Omron CX-Programmer project NewProject (CX-Programmer 9.61)

# PLC Rubber_Sheet_thickness_control: CP1H XA

## Global symbols (name address type ; comment)
0.00 BOOL  ; Autostart
0.01 BOOL  ; Autostop
0.02 BOOL  ; Emergency
0.03 BOOL  ; Automode
0.04 BOOL  ; Emergency
0.10 BOOL  ; HMI1
0.11 BOOL  ; HMI2
0.12 BOOL  ; HMI3
0.13 BOOL  ; HMI4
100.00 BOOL  ; Auto_start_HMI
100.02 BOOL  ; PB_LAMP_GREEN
100.03 BOOL  ; PB_LAMP_RED
100.04 BOOL  ; Tipis_kiri
100.05 BOOL  ; Tebal_kiri
100.06 BOOL  ; Tipis _kanan
100.07 BOOL  ; Tebal_kanan
101.00 BOOL  ; TL_RED
101.01 BOOL  ; TL_YELLOW
101.02 BOOL  ; TL_GREEN
200 CHANNEL  ; Analog input 1
200.00 BOOL  ; Autostart_HMI
200.10 BOOL  ; EMO_AL
201 CHANNEL  ; Analog input 2
C0 CHANNEL  ; TIME
C0000 BOOL  ; COUNTER_1
D0 CHANNEL  ; SET_TIPIS_KIRI
D1 CHANNEL  ; SET_TEBAL_KIRI
D2 CHANNEL  ; SET_TIPIS_KANAN
D300 CHANNEL  ; SET_TEBAL_KANAN
D3010 CHANNEL  ; scalling 2
D310 CHANNEL  ; scalling 2
D400 CHANNEL  ; Output A
D410 CHANNEL  ; output B
D420 CHANNEL  ; output A
D5 CHANNEL  ; Scalled Ouput 0
H0.00 BOOL  ; TIPKIR
H0.01 BOOL  ; TEBKIR
H0.02 BOOL  ; TIPKAN
H0.03 BOOL  ; TEBKAN
H0.04 BOOL  ; TIPIS
H0.05 BOOL  ; TEBAL
H0.09 BOOL  ; TIPIS
H0.10 BOOL  ; TEBAL
H0.11 BOOL  ; HMI_Left thin adjust (button)
H0.12 BOOL  ; HMI_Left thick adjust (button)
H0.13 BOOL  ; HMI_Right thin adjust (button)
H0.14 BOOL  ; HMI_Right thick adjust (button)
H0.15 BOOL  ; reset timer
H100.00 BOOL  ; HOLD_Auto Start
H100.15 BOOL  ; reset timer
H200.01 BOOL  ; EMO_AL
H200.02 BOOL  ; TIPIS
H200.03 BOOL  ; TEBAL
T0000 BOOL  ; TIPKIR
T0001 BOOL  ; TEBKIR
T0002 BOOL  ; TIPKAN
T0003 BOOL  ; TEBKAN
T0004 BOOL  ; TIPIS
T0005 BOOL  ; TEBAL
T0006 BOOL  ; T_LIMIT
T0007 BOOL  ; T_LIMIT
T0008 BOOL  ; T_LIMIT
T0009 BOOL  ; T_LIMIT
T0010 BOOL  ; T_LIMIT
T0011 BOOL  ; T_LIMIT
W0 CHANNEL  ; TIPKIR
W1 CHANNEL  ; TEBKIR
W2 CHANNEL  ; TIPKAN
W3 CHANNEL  ; TEBKAN
W4 CHANNEL  ; TIPIS
W5 CHANNEL  ; TEBAL
W6 CHANNEL  ; TIME

## Program NewProgram1 (cyclic task 0)
Local symbols
TEBAL BOOL

### Section MAIN
; READ SENSOR

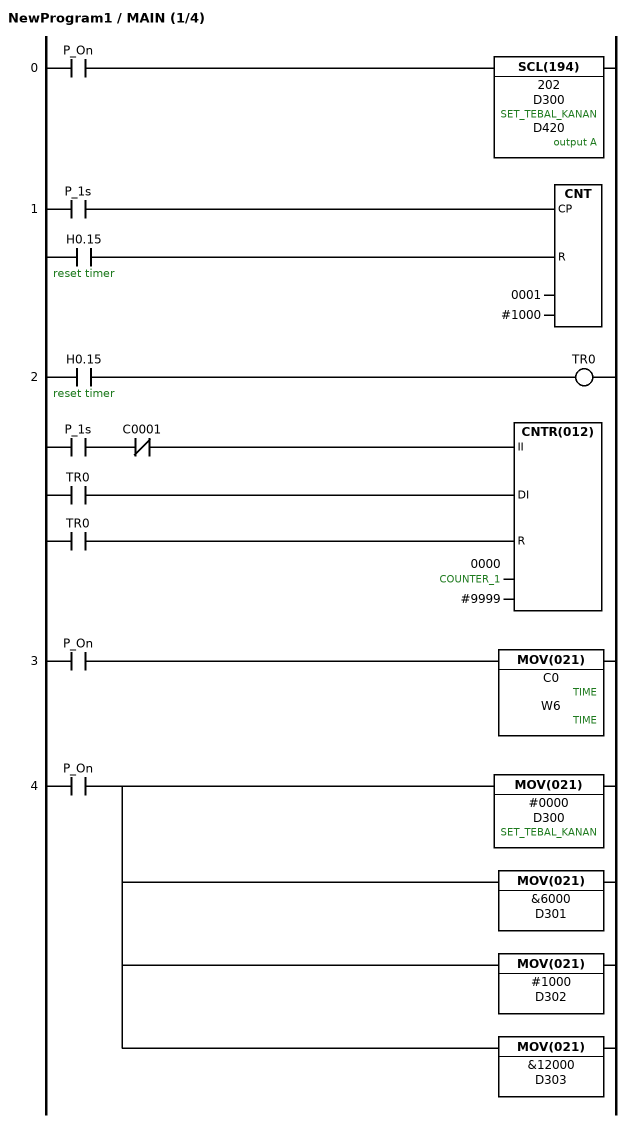
; rung 0
LD P_On
SCL(194) 202 D300 D420  ; SET_TEBAL_KANAN, output A
; rung 1
LD P_1s
LD H0.15  ; reset timer
CNT 0001 #1000
; rung 2
LD P_1s
ANDNOT C0001
LD H0.15  ; reset timer
OUT TR0
LD TR0
CNTR(012) 0000 #9999  ; COUNTER_1
; rung 3
LD P_On
MOV(021) C0 W6  ; TIME
; rung 4
LD P_On
MOV(021) #0000 D300  ; SET_TEBAL_KANAN
MOV(021) &6000 D301
MOV(021) #1000 D302
MOV(021) &12000 D303

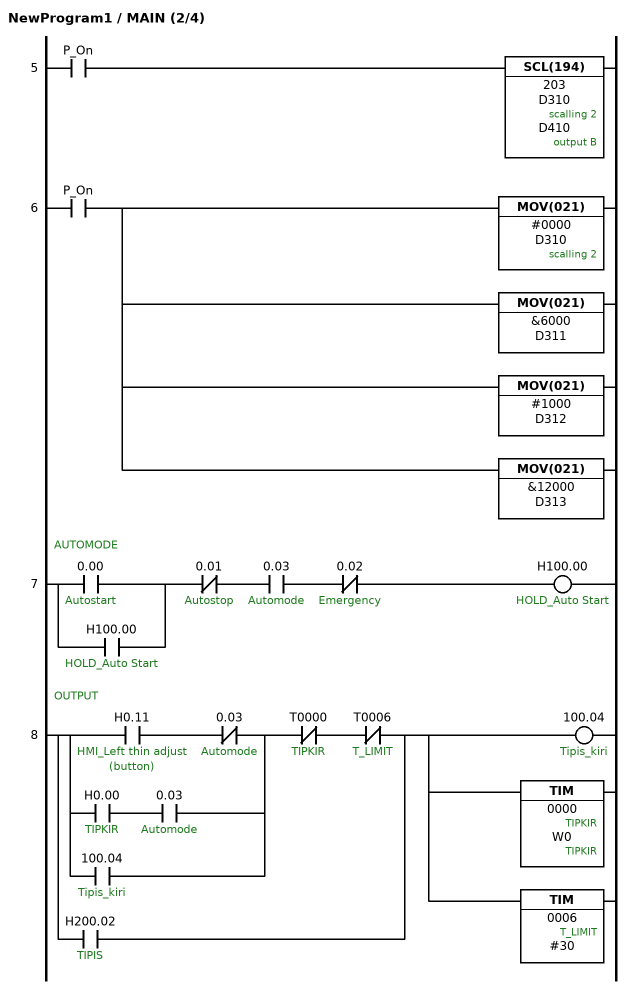
; rung 5
LD P_On
SCL(194) 203 D310 D410  ; scalling 2, output B
; rung 6
LD P_On
MOV(021) #0000 D310  ; scalling 2
MOV(021) &6000 D311
MOV(021) #1000 D312
MOV(021) &12000 D313
; rung 7: AUTOMODE
LD 0.00  ; Autostart
OR H100.00  ; HOLD_Auto Start
ANDNOT 0.01  ; Autostop
AND 0.03  ; Automode
ANDNOT 0.02  ; Emergency
OUT H100.00  ; HOLD_Auto Start
; rung 8: OUTPUT
LD H0.11  ; HMI_Left thin adjust (button)
ANDNOT 0.03  ; Automode
LD H0.00  ; TIPKIR
AND 0.03  ; Automode
ORLD
OR 100.04  ; Tipis_kiri
ANDNOT T0000  ; TIPKIR
ANDNOT T0006  ; T_LIMIT
OR H200.02  ; TIPIS
OUT 100.04  ; Tipis_kiri
TIM 0000 W0  ; TIPKIR
TIM 0006 #30  ; T_LIMIT

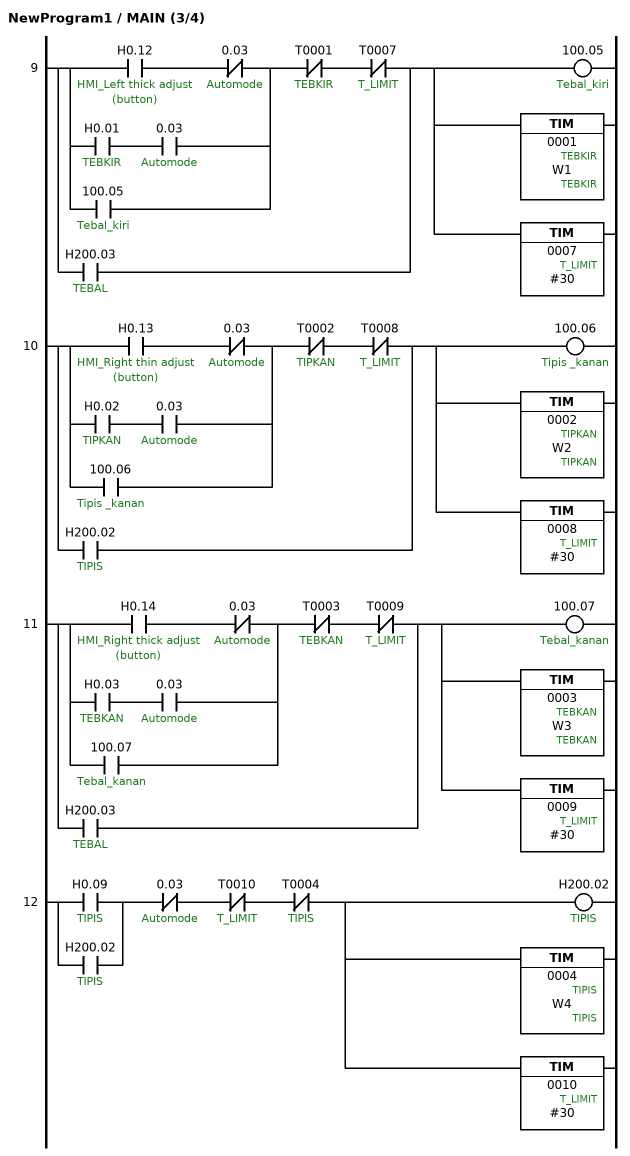
; rung 9
LD H0.12  ; HMI_Left thick adjust (button)
ANDNOT 0.03  ; Automode
LD H0.01  ; TEBKIR
AND 0.03  ; Automode
ORLD
OR 100.05  ; Tebal_kiri
ANDNOT T0001  ; TEBKIR
ANDNOT T0007  ; T_LIMIT
OR H200.03  ; TEBAL
OUT 100.05  ; Tebal_kiri
TIM 0001 W1  ; TEBKIR
TIM 0007 #30  ; T_LIMIT
; rung 10
LD H0.13  ; HMI_Right thin adjust (button)
ANDNOT 0.03  ; Automode
LD H0.02  ; TIPKAN
AND 0.03  ; Automode
ORLD
OR 100.06  ; Tipis _kanan
ANDNOT T0002  ; TIPKAN
ANDNOT T0008  ; T_LIMIT
OR H200.02  ; TIPIS
OUT 100.06  ; Tipis _kanan
TIM 0002 W2  ; TIPKAN
TIM 0008 #30  ; T_LIMIT
; rung 11
LD H0.14  ; HMI_Right thick adjust (button)
ANDNOT 0.03  ; Automode
LD H0.03  ; TEBKAN
AND 0.03  ; Automode
ORLD
OR 100.07  ; Tebal_kanan
ANDNOT T0003  ; TEBKAN
ANDNOT T0009  ; T_LIMIT
OR H200.03  ; TEBAL
OUT 100.07  ; Tebal_kanan
TIM 0003 W3  ; TEBKAN
TIM 0009 #30  ; T_LIMIT
; rung 12
LD H0.09  ; TIPIS
OR H200.02  ; TIPIS
ANDNOT 0.03  ; Automode
ANDNOT T0010  ; T_LIMIT
ANDNOT T0004  ; TIPIS
OUT H200.02  ; TIPIS
TIM 0004 W4  ; TIPIS
TIM 0010 #30  ; T_LIMIT

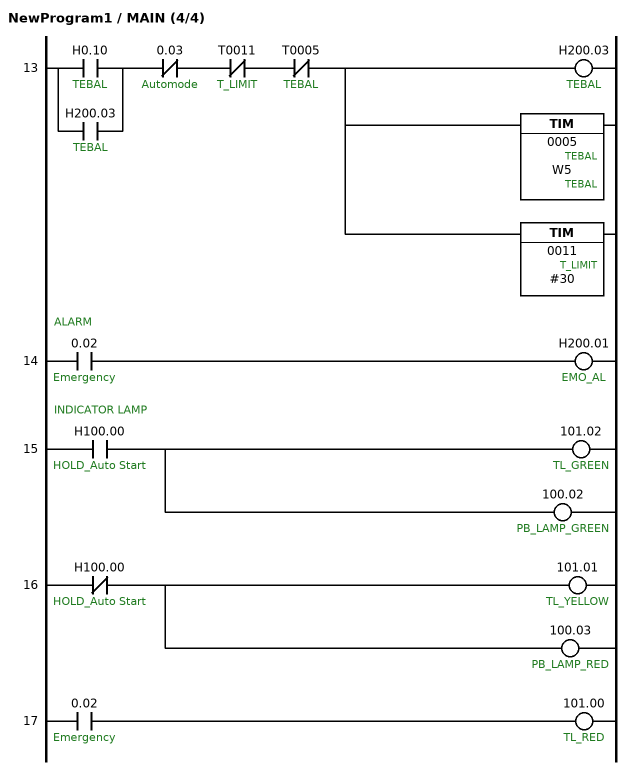
; rung 13
LD H0.10  ; TEBAL
OR H200.03  ; TEBAL
ANDNOT 0.03  ; Automode
ANDNOT T0011  ; T_LIMIT
ANDNOT T0005  ; TEBAL
OUT H200.03  ; TEBAL
TIM 0005 W5  ; TEBAL
TIM 0011 #30  ; T_LIMIT
; rung 14: ALARM
LD 0.02  ; Emergency
OUT H200.01  ; EMO_AL
; rung 15: INDICATOR LAMP
LD H100.00  ; HOLD_Auto Start
OUT 101.02  ; TL_GREEN
OUT 100.02  ; PB_LAMP_GREEN
; rung 16
LDNOT H100.00  ; HOLD_Auto Start
OUT 101.01  ; TL_YELLOW
OUT 100.03  ; PB_LAMP_RED
; rung 17
LD 0.02  ; Emergency
OUT 101.00  ; TL_RED

### Section END
; rung 0
END(001)